{attribute 'GeneratedUsingTerminal: EL5101-0011-0016'}
{attribute addProperty BoxType "EL5101-0011-0016"}
{attribute addProperty Id "EtcSlaveTerminalBaseENC_StatusAT %I*ENC_Status_4E2088B98ENC_NextSync1TimeAT %I*ENC_NextSync1Time_9AFDC2758ENC_TxPdo_1_Samples_Counter_valueAT %I*ENC_TxPdo_1_Samples_Counter_value_215818C64ENC_ControlAT %Q*ENC_Control_14E3EF4F5WcStateAT %I*WcState_9091E0EB2InfoDataAT %I*InfoData_BEF6B88E18"}
{attribute addProperty CRC "816454837"}
{attribute addProperty Size "45"}
TYPE EL5101_30AA1CB5 EXTENDS EtcSlaveTerminalBase :
STRUCT
	{attribute addProperty Name "ENC_Status"}
	ENC_Status : ENC_Status_4E2088B9;
	{attribute addProperty Name "ENC_NextSync1Time"}
	ENC_NextSync1Time : ENC_NextSync1Time_9AFDC275;
	{attribute addProperty Name "ENC_TxPdo_1_Samples_Counter_value"}
	ENC_TxPdo_1_Samples_Counter_value : ENC_TxPdo_1_Samples_Counter_value_215818C6;
	{attribute addProperty Name "ENC_Control"}
	ENC_Control : ENC_Control_14E3EF4F;
	{attribute addProperty Name "WcState"}
	WcState : WcState_9091E0EB;
	{attribute addProperty Name "InfoData"}
	InfoData : InfoData_BEF6B88E;
END_STRUCT
END_TYPE

(* stored: Version 1.2.0.0, ProductVersion 3.1.4024.9
   DUT EL5101_30AA1CB5: Id {da94f99d-c484-4461-9c66-e1afa492b215} *)
